// Master Arm Base Controller, Hold at Current Posture
FUNCTION_BLOCK FB_MasterArmCtrlBase IMPLEMENTS I_MasterArmCtrl
VAR_INPUT
END_VAR
VAR_OUTPUT
END_VAR
VAR
	// flag if the controller has finished all its jobs
	m_isFinished:BOOL:=FALSE;
	
	// controller execute time period
	m_timePeriod :LREAL:=0;
	
	// flag to hold last commands
	m_holdLastCmds :BOOL := FALSE;
	
	// arm control data
	m_cmdJntPos : VEC7d;
	m_cmdJntVel : VEC7d;
	m_cmdJntAcc : VEC7d;
	m_cmdJntTrq : VEC7d;
	m_jntOPMode : Vec7i;
	m_jntEnableFlag :Vec7i;
	m_cmdCartPose : ST_Frame;
	m_cmdCartTwist : Vec6d;
END_VAR

// override this function in each exact controller
METHOD PROTECTED calcCmdJntPos : BOOL

VAR_IN_OUT CONSTANT
	i_slaveIdx :INT;
	i_shoulderPose :ST_Frame;
	i_masterArm :FB_MasterArm;
	i_slaveStatus :ST_SlaveStatus;
END_VAR
END_METHOD

// override this function in each exact controller
METHOD PROTECTED calcCmdJntTrq : BOOL

VAR_IN_OUT CONSTANT
	i_slaveIdx :INT;
	i_shoulderPose :ST_Frame;
	i_masterArm :FB_MasterArm;
	i_slaveStatus :ST_SlaveStatus;
END_VAR
// set joint torque to zero in default
m_cmdJntTrq := g_zeroVec7d;
END_METHOD

METHOD checkToHoldLastCmds : BOOL
VAR_IN_OUT CONSTANT
	i_masterArm :FB_MasterArm;
END_VAR
VAR
	j:INT;
	maxJntErr:LREAL;
	jntCtrlErr:Vec7d;
END_VAR
// check if to hold the command joint position unchanged
vecSub(i_masterArm.m_cmdJntPos, i_masterArm.m_curJntPos,jntCtrlErr);
maxJntErr:=0.0;
FOR j:=1 TO g_mJntNum DO
	maxJntErr:= MAX(maxJntErr, ABS(jntCtrlErr[j]));
END_FOR

checkToHoldLastCmds := (maxJntErr<g_jntCtrlErrForCmdHold);
END_METHOD

METHOD copyCmds : BOOL
VAR_IN_OUT 
	r_masterArmCtrlCmd :ST_ArmCtrlCmds;
END_VAR
r_masterArmCtrlCmd.m_jntEnableFlag :=m_jntEnableFlag;
r_masterArmCtrlCmd.m_cmdCartPose:=m_cmdCartPose;
r_masterArmCtrlCmd.m_cmdCartTwist:=m_cmdCartTwist;
r_masterArmCtrlCmd.m_cmdJntPos:=m_cmdJntPos;
r_masterArmCtrlCmd.m_cmdJntVel:=m_cmdJntVel;
r_masterArmCtrlCmd.m_cmdJntAcc:=m_cmdJntAcc;
r_masterArmCtrlCmd.m_cmdJntTrq:=m_cmdJntTrq;
r_masterArmCtrlCmd.m_jntOPMode:=m_jntOPMode;
END_METHOD

// override this function in each exact controller
// NOTICE: set joint control mode here, and do some initialization if needed
METHOD PUBLIC init : BOOL
VAR_IN_OUT CONSTANT
	i_masterArm	:FB_MasterArm;
END_VAR
VAR_IN_OUT 
	r_masterArmCtrlCmd :ST_ArmCtrlCmds;
END_VAR
m_timePeriod:=0;
m_jntEnableFlag :=g_onesVec7i;
m_jntOPMode:=g_allPosTrqMode;
m_cmdCartPose:=i_masterArm.curCartPose;
m_cmdCartTwist:=g_zeroVec6d;
IF FALSE = m_holdLastCmds THEN
	m_cmdJntPos:=i_masterArm.curJntPos;
ELSE 
	m_cmdJntPos := r_masterArmCtrlCmd.m_cmdJntPos;
END_IF
m_cmdJntVel:=g_zeroVec7d;
m_cmdJntAcc:=g_zeroVec7d;
m_cmdJntTrq:=g_zeroVec7d;

// update commands to arm
copyCmds(r_masterArmCtrlCmd);
END_METHOD

PROPERTY isFinished : BOOL
GET
isFinished:=m_isFinished;
END_GET
END_PROPERTY

{warning '添加方法实现'}
METHOD reset : BOOL
m_isFinished:=FALSE;
END_METHOD

{warning '添加方法实现'}
METHOD run : BOOL

VAR_IN_OUT CONSTANT
	i_slaveIdx :INT;
	i_shoulderPose :ST_Frame;
	i_masterArm :FB_MasterArm;
	i_slaveStatus :ST_SlaveStatus;
END_VAR
VAR_IN_OUT
	r_masterArmCtrlCmd :ST_ArmCtrlCmds;
END_VAR
VAR
	i:INT;
END_VAR
IF m_isFinished THEN
	RETURN;
END_IF

// check if arm enabled
IF FALSE = i_masterArm.isEnabled(m_jntEnableFlag) THEN
	RETURN;
END_IF

// calculate command joint position--Motion control
calcCmdJntPos(i_slaveIdx, i_shoulderPose, i_masterArm,i_slaveStatus);

// calculate command joint torque -- Force control
calcCmdJntTrq(i_slaveIdx, i_shoulderPose, i_masterArm,i_slaveStatus);

// update commands to arm
copyCmds(r_masterArmCtrlCmd);

// update time period
m_timePeriod := m_timePeriod+g_armCtrlCycleTime;
END_METHOD

PROPERTY timePeriod : Lreal
GET
timePeriod := m_timePeriod;
END_GET
END_PROPERTY

END_FUNCTION_BLOCK

(* stored: Version 1.1.0.1, ProductVersion 3.1.4024.11
   POU FB_MasterArmCtrlBase: Id {dee0ec68-3abc-4720-b67c-0fb3fd57933b}, SpecialFunc None
   Method calcCmdJntPos: Id {98ab3239-d030-4534-a55d-1eaac78d6af0}
   Method calcCmdJntTrq: Id {31ee0fe6-80c4-42e7-bd18-5b745e895642}
   Method checkToHoldLastCmds: Id {90f04ad1-6a41-4802-98b4-abd6341aeded}
   Method copyCmds: Id {e9e5f0a1-1fa4-4d4d-889b-b9e9ec07137a}
   Method init: Id {63e02c69-11c3-4e06-9c58-dcaf1b3a881b}
   Property isFinished: Id {d6db4485-2c6d-406e-9b85-5a477e39dd21}
   Get Get: Id {438b47e5-c18c-4fc8-a8d2-2d2ca67eaf31}
   Method reset: Id {ac9e4b6b-f016-4e25-9efd-13892d3b6c48}
   Method run: Id {4a86d5bc-6efe-47db-8e4e-968f76a73eb3}
   Property timePeriod: Id {44038474-1ba7-4c9c-8c84-72a6505c50bc}
   Get Get: Id {a96f8ba3-aad3-45c7-b8fb-41d2e22f00f8} *)
